(* PLC project CoDeSys External Library Template, WAGO e!COCKPIT e!COCKPIT, author 3S - Smart Software Solutions GmbH *)
(* stored: creationDateTime 2019-10-29T12:22:40.3516465, version 3.5.5.30, modificationDateTime 2019-10-24T14:40:07.960949, organization 3S - Smart Software Solutions GmbH *)
(* Library project template with all possible element types, docu and a sample project structure *)

(* Autor: Paweł Kąkol, 2018-08-13-PK Prawa majątkowe: Solwena Sp. z o.o., Aktualizacje: 2018-09-10-PK: dodanie klasy alarmów dla ResetKonwertera i BrakTelegramowEnOcean 2019-02-18-AWy: zmiana klas alarmów Opis: enum służy do definicji klas alarmów w fb konwertera GTW0 na budynkach PPP Sopot *)
{attribute 'qualified_only'}
{attribute 'strict'}
TYPE enumPPPSBramkaSTC65RS485ModbusErrorKlasa : (BrakKomunikacji := enumKlasaAlarmu.AwariaAutomatyki, ResetKonwertera := enumKlasaAlarmu.AwariaAutomatyki, BrakTelegramowEnOcean := enumKlasaAlarmu.AwariaAutomatyki);
END_TYPE
